TYPE ST_CommunicatorStack :
STRUCT
	stMessage					: ST_CommunicatorMassege;
	bSent						: BOOL;		//wysłane
	bConfirmation				: BOOL;		//potwierdzenie
	itfSender					: ITF_MessengerSender;
	itfRecipient				: ITF_MessengerRecipient;
	
END_STRUCT
END_TYPE

(* stored: Version 1.1.0.1
   DUT ST_CommunicatorStack: Id {f3df0a22-2d82-062c-18b5-7c2b5a82b67e} *)
